// TIA Portal V18 export
// export: Created 2025-12-01T12:38:48.977886Z, ExportSetting None, DisplayName Totally Integrated Automation Portal, DisplayVersion V18 Update 5, DisplayName TIA Portal Openness, DisplayVersion V18 Update 5, DisplayName TIA Portal Teamcenter Gateway, DisplayVersion V18, DisplayName TIA Portal Version Control Interface, DisplayVersion V18, DisplayName STEP 7 Professional, DisplayVersion V18 Update 5, DisplayName STEP 7 Safety, DisplayVersion V18, DisplayName WinCC Professional, DisplayVersion V18 Update 5
FUNCTION "CuringOven" : Void   // FC900, LAD
{ S7_Optimized_Access := 'TRUE' }
// stored: AutoNumber false, SetENOAutomatically false
BEGIN

REGION Network 1
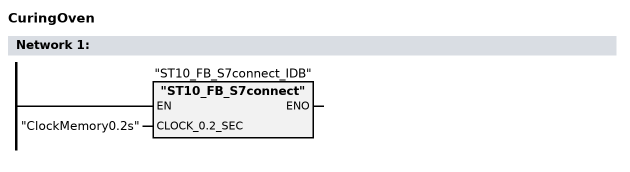
   RUNG wire#powerrail
      "ST10_FB_S7connect_IDB"("CLOCK_0.2_SEC" := "ClockMemory0.2s")
   END_RUNG
   // the same network as SCL:
   "ST10_FB_S7connect_IDB"("CLOCK_0.2_SEC" := "ClockMemory0.2s");   // "ST10_FB_S7connect"
END_REGION
END_FUNCTION
